FUNCTION_BLOCK FB_Step
VAR_IN_OUT
    sm : FB_StateMachine;
END_VAR

VAR_INPUT
    nStep : DINT;
    nNextStep : DINT;
    nTimeout : DINT;
    sName : STRING(80);
END_VAR

VAR_OUTPUT
    Entry : BOOL;
    Execute : BOOL;
    Exiting : BOOL;
END_VAR

VAR
    _perms : FB_Permissives;
    _mappedBits : INT;
    _active : BOOL;
    _prevActive : BOOL;
    _permsSatisfied : BOOL;
    _permsEvalReady : BOOL;
    _exitDone : BOOL;
    _effectiveNextStep : DINT;
    _hasOverride : BOOL;
END_VAR


// Evaluate permissives from previous cycle's MapPerm calls
// Unmapped bits are automatically bypassed (auto-pass)
_perms.cfg.BypassPermissives := NOT _mappedBits;
_perms.cfg.Name := sName;
_perms();
_permsSatisfied := _perms.sts.OK;
_mappedBits := 0;

// Check if this step is the active step in the state machine
_active := (sm.StepInfo.CurrentStep = nStep);

// Default next step unless overridden
IF NOT _hasOverride THEN
    _effectiveNextStep := nNextStep;
END_IF;

// Reset lifecycle outputs each scan
Entry := FALSE;
Execute := FALSE;
Exiting := FALSE;

IF _active THEN
    // Report step metadata to state machine for HMI visibility
    sm.ReportStepInfo(sName := sName, stPerms := _perms.cfg);

    IF NOT _prevActive THEN
        //---------------------------------------------------------------------
        // ENTRY: first scan this step is active
        //---------------------------------------------------------------------
        Entry := TRUE;
        _permsEvalReady := FALSE;
        _exitDone := FALSE;
        _hasOverride := FALSE;

    ELSIF NOT _permsEvalReady THEN
        //---------------------------------------------------------------------
        // First EXECUTE scan: perms are being mapped, eval next cycle
        //---------------------------------------------------------------------
        Execute := TRUE;
        _permsEvalReady := TRUE;

    ELSIF NOT _permsSatisfied THEN
        //---------------------------------------------------------------------
        // EXECUTE: waiting for all mapped permissives to be satisfied
        //---------------------------------------------------------------------
        IF NOT sm.Status.Faulted THEN
            Execute := TRUE;
        END_IF;

        // Timeout fault detection
        IF nTimeout > 0 AND sm.StepInfo.StepTimerSeconds > DINT_TO_REAL(nTimeout) THEN
            sm.SetStepFault(bFault := TRUE);
        END_IF;

    ELSIF NOT _exitDone THEN
        //---------------------------------------------------------------------
        // EXIT: all permissives satisfied, one-scan cleanup
        //---------------------------------------------------------------------
        Exiting := TRUE;
        _exitDone := TRUE;

    ELSE
        //---------------------------------------------------------------------
        // ADVANCE: post-exit, request next step from state machine
        //---------------------------------------------------------------------
        sm.SetNextStep(nStep := _effectiveNextStep);
    END_IF;

ELSE
    // Reset lifecycle tracking when step is not active
    _permsEvalReady := FALSE;
    _exitDone := FALSE;
    _hasOverride := FALSE;
END_IF;

_prevActive := _active;

METHOD MapPerm
VAR_INPUT
    nIndex : INT;
    sDescription : STRING;
    bValue : BOOL;
END_VAR
_perms.MapReason(nIndex := nIndex, sDescription := sDescription, bValue := bValue);
IF nIndex >= 0 AND nIndex <= 15 THEN
    _mappedBits := _mappedBits OR SHL(INT#1, nIndex);
END_IF;
END_METHOD

METHOD SetNextStep
VAR_INPUT
    nStep : DINT;
END_VAR
_effectiveNextStep := nStep;
_hasOverride := TRUE;
END_METHOD

END_FUNCTION_BLOCK

(* stored: Version 1.1.0.1, ProductVersion 3.1.4026.12
   POU FB_Step: Id {a1b2c3d4-e5f6-7890-abcd-ef1234567890}, SpecialFunc None
   Method MapPerm: Id {b2c3d4e5-f6a7-8901-bcde-f12345678901}
   Method SetNextStep: Id {c3d4e5f6-a7b8-9012-cdef-123456789012} *)
